{attribute 'qualified_only'}
{attribute 'strict'}
TYPE MY_ENUM :
(
	ENUM_VALUE_0 := 0,
	ENUM_VALUE_1 := 1
);
END_TYPE

(* stored: Version 1.1.0.1, ProductVersion 3.1.4022.18
   EnumerationTextList DUT: Id {c330bdc9-df70-4edf-8ae2-c8f56d976d70} *)
